(* PLC project MQTT, Beckhoff Automation GmbH TwinCAT PLC Control 3.5.13.20 *)
(* stored: creationDateTime 2021-01-27T09:57:50.4520333, modificationDateTime 2021-01-27T09:57:50.4568417 *)

(* global variable list GVL_MQTT *)
{attribute 'qualified_only'}
VAR_GLOBAL

	mqtt_port: UINT := 1883;
	mqtt_broker: STRING := 'letto.htlwrn.ac.at';
	username: STRING := 'el_mb_bek1';
	password: STRING := 'JsonIsCool';
	mqtt_interval: TIME := T#1S;
END_VAR
